PROGRAM PRG_Main
VAR
	//ADS
	FB_AdsDeviceAPI_1 : FB_AdsCommandRouter;
	FB_AdsDeviceAPI_2 : FB_AdsCommandRouter;
	FB_AdsDeviceAPI_3 : FB_AdsCommandRouter;
	
	//FlowMeter
	AlicatFlowMeter_1: FB_AlicatFlowMeter;
	bConnectToAlicatFlow1: BOOL;
	bRes_AlicatFlowConnected1: BOOL;
	bGetPressureFlow1: BOOL;
	bGetPressureSuccessfulFlow1: BOOL;
	bGetAlicatDataFlow1: BOOL;
	bGetAlicatDataSuccessfulFlow1: BOOL;
	bLockDisplayFlow1: BOOL;
	bLockDisplaySuccessfulFlow1: BOOL;
	bUnlockDisplayFlow1: BOOL;
	bUnlockDisplaySuccessfulFlow1: BOOL;
	bDisconnectFromAlicatFlow1: BOOL;
	bRes_AlicatFlowDisConnected1: BOOL;
	
	AlicatFlowMeter_2 : FB_AlicatFlowMeter;
	AlicatFlowMeter_3 : FB_AlicatFlowMeter;
	AlicatFlowMeter_4 : FB_AlicatFlowMeter;
	
	AlicatAbs_1 : FB_AlicatAbsolute;
	bConnectToAlicatAbs1: BOOL;
	bRes_AlicatAbsConnected1: BOOL;
	bGetPressureAbs1: BOOL;
	bGetPressureSuccessfulAbs1: BOOL;
	bGetAlicatDataAbs1: BOOL;
	bGetAlicatDataSuccessfulAbs1: BOOL;
	bLockDisplayAbs1: BOOL;
	bLockDisplaySuccessfulAbs1: BOOL;
	bUnlockDisplayAbs1: BOOL;
	bUnlockDisplaySuccessfulAbs1: BOOL;
	bDisconnectFromAlicatAbs1: BOOL;
	bRes_AlicatAbsDisConnected1: BOOL;
	
	AlicatAbs_2 : FB_AlicatAbsolute;

	AlicatDiff_1 : FB_AlicatDifferential;
	bConnectToAlicatDiff1: BOOL;
	bRes_AlicatDiffConnected1: BOOL;
	bGetPressureDiff1: BOOL;
	bGetPressureSuccessfulDiff1: BOOL;
	bGetAlicatDataDiff1: BOOL;
	bGetAlicatDataSuccessfulDiff1: BOOL;
	bLockDisplayDiff1: BOOL;
	bLockDisplaySuccessfulDiff1: BOOL;
	bUnlockDisplayDiff1: BOOL;
	bUnlockDisplaySuccessfulDiff1: BOOL;
	bDisconnectFromAlicatDiff1: BOOL;
	bRes_AlicatDiffDisConnected1: BOOL;
	
	AlicatDiff_2 : FB_AlicatDifferential;
	AlicatDiff_3 : FB_AlicatDifferential;
	AlicatDiff_4 : FB_AlicatDifferential;

	//Agilent Vacuum Gauge		
	AgilentVacuum_1 : FB_AgilentVacuumGauge;
	bConnectToAgilentVac: BOOL;
	bRes_AgilentVacConnected: BOOL;
	bGetPressureAgilent: BOOL;
	bGetPressureSuccessfulAgilent: BOOL;
	bDisconnectFromAgilent: BOOL;
	bRes_AgilentDisConnected: BOOL;
	
	//Alicat Flow Meter Return Variables
	AlicatFlowMeterPressure : LREAL; //M_GetPressure
	AlicatFlowDataPressure  : LREAL; //M_GetAlicatFlowData
	AlicatFlowDataTotFlow   : LREAL;
	AlicatFlowMassFlowRate  : LREAL;
	AlicatFlowVolFlowRate   : LREAL;
	
	//AlicatAbs Return Values
	AlicatAbsPressure : LREAL;
	
	//AlicatDiff Return Values
	AlicatDiffPressure : LREAL;
	
	//Agilent Return Values
	AgilentPressure : LREAL;
	
	
	
	
	
	
	
	
	//	bTestInput: BOOL;
//	bTestOutput: BOOL;
//	fbMachine: FB_ExampleMachine;
//	fbStation1: FB_ExampleStation;
//	fbStation2: FB_ExampleStation;
//	fbStation3: FB_ExampleStation;
//	fbStation4: FB_ExampleStation;
//	bStart: BOOL;
//	bAbort: BOOL;
//	bReset: BOOL;
//	bStop: BOOL;
//	bSuspend: BOOL;
//	fbDevice1: FB_ExampleDevice;
//	fbDevice2: FB_ExampleDevice;
//	fbDevice3: FB_ExampleDevice;
//	fbDevice4: FB_ExampleDevice;
//	bPoweredOn: BOOL;	
//	bTestADSServer: BOOL;
//	strTarget: T_MaxString;
//	strCommand: T_MaxString;
//	arrParams: T_ApiMethodParameters;
//	MyResults: T_MaxString;
//	bInterfaceTest : BOOL;
	
END_VAR

A_Machine();

//Alicat Flow Meter 1
IF bConnectToAlicatFlow1 THEN
	bRes_AlicatFlowConnected1 := AlicatFlowMeter_1.M_Connect();
	IF 	bRes_AlicatFlowConnected1 THEN
		bConnectToAlicatFlow1 := FALSE;
	ELSIF AlicatFlowMeter_1.P_bError THEN
		bConnectToAlicatFlow1 := FALSE;
		AlicatFlowMeter_1.M_ClearError();
	END_IF
END_IF

IF bGetAlicatDataFlow1 THEN
	bGetAlicatDataSuccessfulFlow1 := AlicatFlowMeter_1.M_GetAlicatFlowData(_out_lrealPressure=>AlicatFlowDataPressure,
																			 _out_lrealTotFlow=>AlicatFlowDataTotFlow,
																			 _out_lrealMassFlowRate=>AlicatFlowMassFlowRate,
																			 _out_lrealVolFlowRate=>AlicatFlowVolFlowRate);
	IF bGetAlicatDataSuccessfulFlow1 THEN
		bGetAlicatDataFlow1 := FALSE;
	ELSIF AlicatFlowMeter_1.P_bError THEN
		bGetAlicatDataFlow1 := FALSE;
		AlicatFlowMeter_1.M_ClearError();
	END_IF
END_IF

IF bDisconnectFromAlicatFlow1 THEN
	bRes_AlicatFlowDisConnected1 := AlicatFlowMeter_1.M_Disconnect();
	IF bRes_AlicatFlowDisConnected1 THEN
		bDisconnectFromAlicatFlow1 := FALSE;
	ELSIF AlicatFlowMeter_1.P_bError THEN
		bDisconnectFromAlicatFlow1 := FALSE;
		AlicatFlowMeter_1.M_ClearError();
	END_IF
END_IF

IF bGetPressureFlow1 THEN
	bGetPressureSuccessfulFlow1 := AlicatFlowMeter_1.M_GetPressure(_out_lrealPressure => AlicatFlowMeterPressure);
	IF bGetPressureSuccessfulFlow1 THEN		
		bGetPressureFlow1 := FALSE;
	ELSIF AlicatFlowMeter_1.P_bError THEN
		bGetPressureFlow1 := FALSE;
		AlicatFlowMeter_1.M_ClearError();
	END_IF
END_IF

IF bLockDisplayFlow1 THEN
	bLockDisplaySuccessfulFlow1 := AlicatFlowMeter_1.M_LockDisplay();
	IF bLockDisplaySuccessfulFlow1 THEN
		bLockDisplayFlow1 := FALSE;
	ELSIF AlicatFlowMeter_1.P_bError THEN
		bLockDisplayFlow1 := FALSE;
		AlicatFlowMeter_1.M_ClearError();
	END_IF
END_IF

IF bUnlockDisplayFlow1 THEN
	bUnlockDisplaySuccessfulFlow1 := AlicatFlowMeter_1.M_UnlockDisplay();
	IF bUnlockDisplaySuccessfulFlow1 THEN
		bUnlockDisplayFlow1 := FALSE;
	ELSIF AlicatFlowMeter_1.P_bError THEN
		bUnlockDisplayFlow1 := FALSE;
		AlicatFlowMeter_1.M_ClearError();
	END_IF
END_IF

//Alicat Absolute 1

IF bConnectToAlicatAbs1 THEN
	bRes_AlicatAbsConnected1 := AlicatAbs_1.M_Connect();
	IF 	bRes_AlicatAbsConnected1 THEN
		bConnectToAlicatAbs1 := FALSE;
	ELSIF AlicatAbs_1.P_bError THEN
		bConnectToAlicatAbs1 := FALSE;
		AlicatAbs_1.M_ClearError();
	END_IF
END_IF

IF bGetAlicatDataAbs1 THEN
	bGetAlicatDataSuccessfulAbs1 := AlicatAbs_1.M_GetAlicatAbsData();
	IF bGetAlicatDataSuccessfulAbs1 THEN
		bGetAlicatDataAbs1 := FALSE;
	ELSIF AlicatAbs_1.P_bError THEN
		bGetAlicatDataAbs1 := FALSE;
		AlicatAbs_1.M_ClearError();
	END_IF
END_IF

IF bDisconnectFromAlicatAbs1 THEN
	bRes_AlicatAbsDisConnected1 := AlicatAbs_1.M_Disconnect();
	IF bRes_AlicatAbsDisConnected1 THEN
		bDisconnectFromAlicatAbs1 := FALSE;
	ELSIF AlicatAbs_1.P_bError THEN
		bDisconnectFromAlicatAbs1 := FALSE;
		AlicatAbs_1.M_ClearError();
	END_IF
END_IF

IF bGetPressureAbs1 THEN
	bGetPressureSuccessfulAbs1 := AlicatAbs_1.M_GetPressure(_out_lrealPressure=>AlicatAbsPressure);
	IF bGetPressureSuccessfulAbs1 THEN
		bGetPressureAbs1 := FALSE;
	ELSIF AlicatAbs_1.P_bError THEN
		bGetPressureAbs1 := FALSE;
		AlicatAbs_1.M_ClearError();
	END_IF
END_IF

IF bLockDisplayAbs1 THEN
	bLockDisplaySuccessfulAbs1 := AlicatAbs_1.M_LockDisplay();
	IF bLockDisplaySuccessfulAbs1 THEN
		bLockDisplayAbs1 := FALSE;
	ELSIF AlicatAbs_1.P_bError THEN
		bLockDisplayAbs1 := FALSE;
		AlicatAbs_1.M_ClearError();
	END_IF
END_IF

IF bUnlockDisplayAbs1 THEN
	bUnlockDisplaySuccessfulAbs1 := AlicatAbs_1.M_UnlockDisplay();
	IF bUnlockDisplaySuccessfulAbs1 THEN
		bUnlockDisplayAbs1 := FALSE;
	ELSIF AlicatAbs_1.P_bError THEN
		bUnlockDisplayAbs1 := FALSE;
		AlicatAbs_1.M_ClearError();
	END_IF
END_IF

//Alicat Differential 1

IF bConnectToAlicatDiff1 THEN
	bRes_AlicatDiffConnected1 := AlicatDiff_1.M_Connect();
	IF 	bRes_AlicatDiffConnected1 THEN
		bConnectToAlicatDiff1 := FALSE;
	ELSIF AlicatDiff_1.P_bError THEN
		bConnectToAlicatDiff1 := FALSE;
		AlicatDiff_1.M_ClearError();
	END_IF
END_IF

IF bGetAlicatDataDiff1 THEN
	bGetAlicatDataSuccessfulDiff1 := AlicatDiff_1.M_GetAlicatDiffData();
	IF bGetAlicatDataSuccessfulDiff1 THEN
		bGetAlicatDataDiff1 := FALSE;
	ELSIF AlicatDiff_1.P_bError THEN
		bGetAlicatDataDiff1 := FALSE;
		AlicatDiff_1.M_ClearError();
	END_IF
END_IF

IF bDisconnectFromAlicatDiff1 THEN
	bRes_AlicatDiffDisConnected1 := AlicatDiff_1.M_Disconnect();
	IF bRes_AlicatDiffDisConnected1 THEN
		bDisconnectFromAlicatDiff1 := FALSE;
	ELSIF AlicatDiff_1.P_bError THEN
		bDisconnectFromAlicatDiff1 := FALSE;
		AlicatDiff_1.M_ClearError();
	END_IF
END_IF

IF bGetPressureDiff1 THEN
	bGetPressureSuccessfulDiff1 := AlicatDiff_1.M_GetPressure(_out_lrealPressure=>AlicatDiffPressure);
	IF bGetPressureSuccessfulDiff1 THEN
		bGetPressureDiff1 := FALSE;
	ELSIF AlicatDiff_1.P_bError THEN
		bGetPressureDiff1 := FALSE;
		AlicatDiff_1.M_ClearError();
	END_IF
END_IF

IF bLockDisplayDiff1 THEN
	bLockDisplaySuccessfulDiff1 := AlicatDiff_1.M_LockDisplay();
	IF bLockDisplaySuccessfulDiff1 THEN
		bLockDisplayDiff1 := FALSE;
	ELSIF AlicatDiff_1.P_bError THEN
		bLockDisplayDiff1 := FALSE;
		AlicatDiff_1.M_ClearError();
	END_IF
END_IF

IF bUnlockDisplayDiff1 THEN
	bUnlockDisplaySuccessfulDiff1 := AlicatDiff_1.M_UnlockDisplay();
	IF bUnlockDisplaySuccessfulDiff1 THEN
		bUnlockDisplayDiff1 := FALSE;
	ELSIF AlicatDiff_1.P_bError THEN
		bUnlockDisplayDiff1 := FALSE;
		AlicatDiff_1.M_ClearError();
	END_IF
END_IF

IF bConnectToAgilentVac THEN
	bRes_AgilentVacConnected := AgilentVacuum_1.M_Connect();
	IF 	bRes_AgilentVacConnected THEN
		bConnectToAgilentVac := FALSE;
	ELSIF AgilentVacuum_1.P_bError THEN
		bConnectToAgilentVac := FALSE;
		AgilentVacuum_1.M_ClearError();
	END_IF
END_IF

IF bGetPressureAgilent THEN
	bGetPressureSuccessfulAgilent := AgilentVacuum_1.M_GetPressure(_out_lrealPressure=>AgilentPressure);
	IF bGetPressureSuccessfulAgilent THEN
		bGetPressureAgilent := FALSE;
	ELSIF AgilentVacuum_1.P_bError THEN
		bGetPressureAgilent := FALSE;
		AgilentVacuum_1.M_ClearError();
	END_IF
END_IF

IF bDisconnectFromAgilent THEN
	bRes_AgilentDisConnected := AgilentVacuum_1.M_Disconnect();
	IF bRes_AgilentDisConnected THEN
		bDisconnectFromAgilent := FALSE;
	ELSIF AgilentVacuum_1.P_bError THEN
		bDisconnectFromAgilent := FALSE;
		AgilentVacuum_1.M_ClearError();
	END_IF
END_IF

ACTION A_Machine:
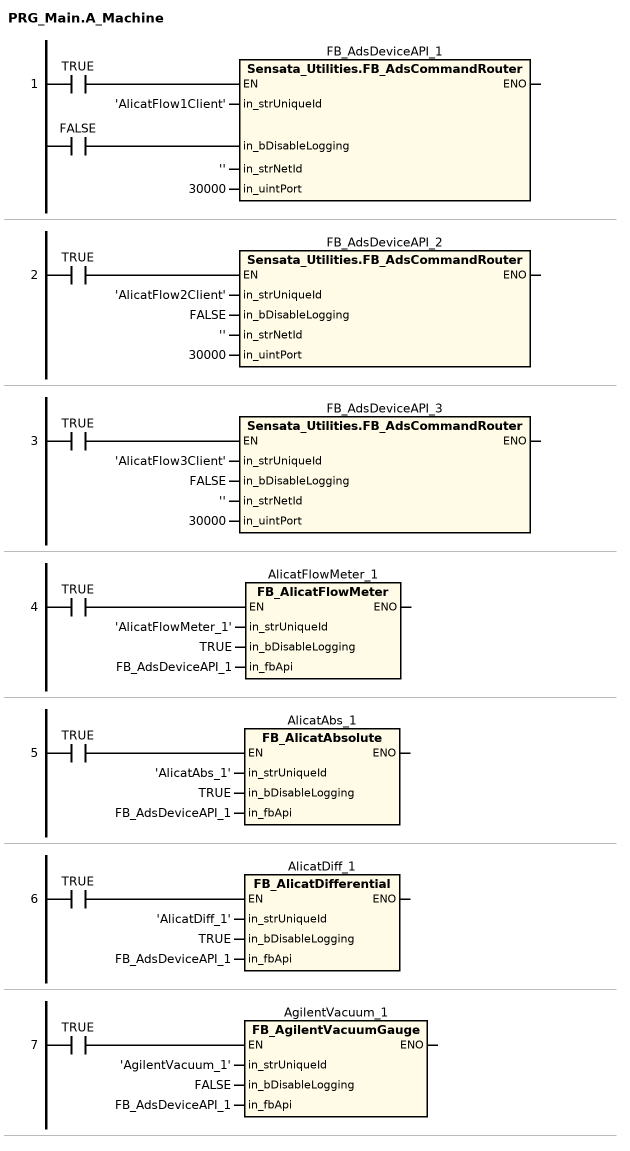
// NETWORK 1
FB_AdsDeviceAPI_1(
    in_strUniqueId := 'AlicatFlow1Client',
    in_bDisableLogging := FALSE,
    in_strNetId := '',
    in_uintPort := 30000); // Sensata_Utilities.FB_AdsCommandRouter

// NETWORK 2
FB_AdsDeviceAPI_2(
    in_strUniqueId := 'AlicatFlow2Client',
    in_bDisableLogging := FALSE,
    in_strNetId := '',
    in_uintPort := 30000); // Sensata_Utilities.FB_AdsCommandRouter

// NETWORK 3
FB_AdsDeviceAPI_3(
    in_strUniqueId := 'AlicatFlow3Client',
    in_bDisableLogging := FALSE,
    in_strNetId := '',
    in_uintPort := 30000); // Sensata_Utilities.FB_AdsCommandRouter

// NETWORK 4
AlicatFlowMeter_1(
    in_strUniqueId := 'AlicatFlowMeter_1',
    in_bDisableLogging := TRUE,
    in_fbApi := FB_AdsDeviceAPI_1); // FB_AlicatFlowMeter

// NETWORK 5
AlicatAbs_1(in_strUniqueId := 'AlicatAbs_1', in_bDisableLogging := TRUE, in_fbApi := FB_AdsDeviceAPI_1); // FB_AlicatAbsolute

// NETWORK 6
AlicatDiff_1(in_strUniqueId := 'AlicatDiff_1', in_bDisableLogging := TRUE, in_fbApi := FB_AdsDeviceAPI_1); // FB_AlicatDifferential

// NETWORK 7
AgilentVacuum_1(
    in_strUniqueId := 'AgilentVacuum_1',
    in_bDisableLogging := FALSE,
    in_fbApi := FB_AdsDeviceAPI_1); // FB_AgilentVacuumGauge
END_ACTION

END_PROGRAM

(* stored: Version 1.1.0.1, ProductVersion 3.1.4024.11
   POU PRG_Main: Id {b13f0be3-4c97-4edc-94e2-8c6f67cb8665}, SpecialFunc None
   Action A_Machine: Id {f2ef6f5c-8a40-4c62-8311-b3186050d362} *)
